Staubli VAL3: Control_Left.pgx

program Control_Left(string& x_sLeftList[])
  local num l_nIndex
begin

  //在屏幕左边进行显示
  //左边的x_sLeftList 是显示的字符串数组

  setTextMode(0)
  //左边栏进行显示
  for l_nIndex=0 to min(7,size(x_sLeftList)-1)
    gotoxy(1,l_nIndex+4)
    if size(x_sLeftList)>l_nIndex and x_sLeftList[l_nIndex]!=""
      put("F"+toString("",l_nIndex+1)+"->"+x_sLeftList[l_nIndex])
    endIf
  endFor
end
